// TwinCAT 3 PLC project PLC
// ProgramVersion: 3.1.4023.0
// libraries:
//   Tc2_MC2, * (Beckhoff Automation GmbH)
//   Tc2_Standard, * (Beckhoff Automation GmbH)
//   Tc2_System, * (Beckhoff Automation GmbH)
//   Tc3_Module, * (Beckhoff Automation GmbH)
//   VisuSymbols,3.5.10.0,System
// project tree:
//   DUTs/ E_Axis.TcDUT, E_MachineState.TcDUT, E_Speed.TcDUT, ST_ErrorData.TcDUT
//   / GlobalTextList.TcGTLO, PlcTask.TcTTO, Visualization Manager.TcVMO (not stored), VISU_TASK.TcTTO
//   GVLs/ GVL.TcGVL
//   POUs/ FB_Machine.TcPOU, FB_Tower.TcPOU, F_HeaderErrorMessage.TcPOU, F_NcErrorMessage.TcPOU, MAIN.TcPOU
//   VISUs/ Tower1.TcVIS
// real-time tasks:
//   TASK PlcTask: cycle T#10ms, priority 20, ADS port 350
//   TASK VISU_TASK: cycle T#200000us, priority 30, ADS port 351
// motion (NC):
//   TASK NC-Task 1 SAF: cycle T#2ms, priority 4, ADS port 501
//   TASK NC-Task 1 SVB: cycle T#10ms, priority 8, ADS port 511
//   AXIS Axis 1 (id 1)
//     General: UnitName=m
//     Dynamic: AccelerationMaximum=1.5, DecelerationMaximum=1.5, Acceleration=1.5, Deceleration=1.5, Jerk=2.25
//     Velo: RefSearch=0.03, RefSync=0.03, SlowManual=0.1, FastManual=1, Maximum=0.1
//     OtherSettings: AllowMotionCmdToSlave=true, PulseDistancePos=0.005, PulseDistanceNeg=0.005
//     encoder EncType=1
//       EncPara: ScaleFactorNumerator=4.166666667e-06, ReferenceSystem=1
//         SoftEndMinControl: Enable=true
//         SoftEndMaxControl: Enable=true, Range=1.44
//         TimeComp: TimeCompMode=1, EncDelayCycles=4
//     drive DrvType=5
//       Analog: VeloReferenz=0.416666666666667, TorqueSetpointScale=10, ScaleFactorActTorque=0.1
//       TimeComp: TaskDelayCycles=1
//     controller CtrType=1
//       CtrPara: PriorControlFactor=1
//         Observer: BandWidth=20
// I/O:
//   DEVICE Device 1 (EtherCAT) (disabled), AmsNetId 192.168.100.90.2.1
//     Drive 1 (N5-2-1) [N5 EtherCAT Drive (CoE)]
// variable links:
//   __THIS__ <-> PLC/PLC Instance
//     Inputs/FromPlc <-> PlcTask Outputs/MAIN.Machine.Tower.stAxis.PlcToNc
//     Outputs/ToPlc <-> PlcTask Inputs/MAIN.Machine.Tower.stAxis.NcToPlc
//   __THIS__ <-> Device 1 (EtherCAT)/Drive 1 (N5-2-1)
//     Drive/Inputs/In/nState1 <-> Transmit PDO 1 Mapping Parameter/Statusword
//     Drive/Inputs/In/nState2 <-> Transmit PDO 1 Mapping Parameter/Statusword @bit 8
//     Drive/Inputs/In/nState4 @bit 1 <-> WcState/InputToggle
//     Drive/Inputs/In/nState4 <-> WcState/WcState
//     Drive/Inputs/In/nState5 <-> Transmit PDO 1 Mapping Parameter/Modes of operation display
//     Drive/Outputs/Out/nCtrl1 <-> Receive PDO 1 Mapping Parameter/Controlword
//     Drive/Outputs/Out/nCtrl2 <-> Receive PDO 1 Mapping Parameter/Controlword @bit 8
//     Drive/Outputs/Out/nCtrl5 <-> Receive PDO 1 Mapping Parameter/Modes of operation
//     Drive/Outputs/Out/nDataOut1 <-> Receive PDO 1 Mapping Parameter/Target Position
//     Enc/Inputs/In/nDataIn1 <-> Transmit PDO 1 Mapping Parameter/Position actual value
//     Enc/Inputs/In/nState4 @bit 1 <-> WcState/InputToggle
//     Enc/Inputs/In/nState4 <-> WcState/WcState
//   NC-Task 1 SAF/Axes/Axis 1 <-> PLC/PLC Instance
//     Inputs/FromPlc <-> PlcTask Outputs/MAIN.Machine.Tower.stAxis.PlcToNc
//     Outputs/ToPlc <-> PlcTask Inputs/MAIN.Machine.Tower.stAxis.NcToPlc

CONFIGURATION PLC
    RESOURCE PLC ON TwinCAT3
        TASK PlcTask(INTERVAL := T#10ms, PRIORITY := 20);
        TASK VISU_TASK(INTERVAL := T#200000us, PRIORITY := 30);
        PROGRAM MAIN WITH PlcTask : MAIN;
        PROGRAM VisuElems_Visu_Prg WITH VISU_TASK : VisuElems.Visu_Prg;
    END_RESOURCE
END_CONFIGURATION

// ---- DUTs/E_Axis.TcDUT
{attribute 'qualified_only'}
{attribute 'strict'}
{attribute 'to_string'}
TYPE E_Axis :
(
	Disabled,
	Enabled,
	Idle,
	MoveAbs,
	Stop,
	Error,
	Reset,
	ManualMode
);
END_TYPE

// ---- DUTs/E_MachineState.TcDUT
{attribute 'qualified_only'}
{attribute 'strict'}
{attribute 'to_string'}
TYPE E_MachineState :
(
	Error,
	Ready,
	Running
);
END_TYPE

// ---- DUTs/E_Speed.TcDUT
{attribute 'qualified_only'}
{attribute 'strict'}
{attribute 'to_string'}
TYPE E_Speed :
(
	Low,
	High
);
END_TYPE

// ---- DUTs/ST_ErrorData.TcDUT
TYPE ST_ErrorData :
STRUCT
	nErrorID			: UDINT;
	sTimeStamp			: STRING;
	sErrorMessageBody	: STRING[300];
	sErrorMessageHeader	: STRING[300];	
	eLastState			: E_Axis;
END_STRUCT
END_TYPE

// ---- GVLs/GVL.TcGVL
VAR_GLOBAL

	eMachineState					: E_MachineState;
	UI_EnableHighSpeed				: BOOL;
END_VAR

// ---- POUs/MAIN.TcPOU
PROGRAM MAIN
VAR
	Machine : FB_Machine; 
	
END_VAR

Machine();

END_PROGRAM

// ---- POUs/FB_Machine.TcPOU
FUNCTION_BLOCK FB_Machine
VAR_INPUT
END_VAR
VAR_OUTPUT

END_VAR
VAR
	Tower : FB_Tower;
	//fManualLowSpeed		: LREAL;
	//fManualHighSpeed	: LREAL;	
	
END_VAR

Tower();

(*
MCJog( Axis := 	stAxis, Velocity := fManualVelocity, Mode := MC_JOGMODE_CONTINOUS );				
McPower(Axis := stAxis);
McReset(Axis := stAxis); 
ActUpdateAxisData();
ActUpdateManVelocity();


CASE GVL.eMachineState OF
	

	// The machine starts up in Error state
	E_MachineState.Error:	
	
	// Changes statet to Ready state
	IF startButton THEN
		readyLamp := TRUE;
		SetState( E_MachineState.Ready );
	END_IF
	
	
	
	E_MachineState.Ready:
	McReset.Execute := TRUE;
		IF McReset.Done THEN 
			McReset.Execute := FALSE; 
		END_IF 	
	
		IF (ActualPos < lowerLimit OR ActualPos > upperLimit) AND enableButton THEN
			 
			IF ActualPos > upperLimit AND enableButton THEN
				McPower.Enable 			:= TRUE;
				McPower.Enable_Negative := TRUE;
				SetState( E_MachineState.Running );
			END_IF
			
			IF ActualPos < lowerLimit AND enableButton THEN 
				McPower.Enable 			:= TRUE;
				McPower.Enable_Positive := TRUE;
				SetState( E_MachineState.Running );
			END_IF
		END_IF
		
 		// Enables the axis for movement
		IF enableButton AND ActualPos > lowerLimit AND ActualPos < upperLimit  THEN
			McPower.Enable 			:= TRUE;
			McPower.Enable_Positive := TRUE; 
			McPower.Enable_Negative := TRUE;		
			SetState( E_MachineState.Running );
		END_IF
		
		// Disables the axis for movement
		IF stopButton THEN
			McPower.Enable 			:= FALSE;
			McPower.Enable_Positive := FALSE; 
			McPower.Enable_Negative := FALSE;
			enableButton 			:= FALSE;
			MCJog.JogForward 		:= FALSE; 
			MCJog.JogBackwards 		:= FALSE;
		END_IF
			
			
	E_MachineState.Running: 	
		
		// forward and backward movement logic
		IF forwardButton OR backwardButton THEN
			IF (ActualPos > lowerLimit AND ActualPos < upperLimit) THEN 
				McPower.Enable_Positive := TRUE; 
				McPower.Enable_Negative := TRUE;
			END_IF 
			IF forwardButton THEN 
				MCJog.JogForward 	:= TRUE;
				MCJog.JogBackwards 	:= FALSE;
			END_IF 
			
			IF backwardButton THEN
				MCJog.JogBackwards 	:= TRUE; 
				MCJog.JogForward 	:= FALSE;
			END_IF 
		ELSE 
			MCJog.JogBackwards 	:= FALSE;
			MCJog.JogForward 	:= FALSE;
		END_IF
		
		// Disables the axis for movement
		IF stopButton THEN
			McPower.Enable 			:= FALSE;
			McPower.Enable_Positive := FALSE; 
			McPower.Enable_Negative := FALSE;
			enableButton 			:= FALSE;
			MCJog.JogForward 		:= FALSE; 
			MCJog.JogBackwards 		:= FALSE;
	
			SetState( E_MachineState.Ready );
		END_IF  
		
		IF (ActualPos < lowerLimit OR ActualPos > upperLimit) AND McPower.Enable_Positive AND McPower.Enable_Negative THEN 
			McPower.Enable 			:= FALSE;
			McPower.Enable_Positive := FALSE; 
			McPower.Enable_Negative := FALSE;
			enableButton 			:= FALSE;
			MCJog.JogForward 		:= FALSE; 
			MCJog.JogBackwards 		:= FALSE;
	
			SetState( E_MachineState.Error );
		END_IF
		

END_CASE

*)

END_FUNCTION_BLOCK

// ---- POUs/FB_Tower.TcPOU

FUNCTION_BLOCK FB_Tower
VAR_INPUT
	resetButton			: BOOL;
	startButton			: BOOL;
	stopButton 			: BOOL;
	forwardButton 		: BOOL; 
	backwardButton 		: BOOL;
	fManualVelocity		: LREAL;
	
	// velocity constant for HIGH and LOW value. 
	fManualLowSpeed		: LREAL := 0.05;
	fManualHighSpeed	: LREAL := 0.1;	
END_VAR
VAR_OUTPUT
END_VAR
VAR
	// Libraries used
	stAxis 				: AXIS_REF;
	MCJog 				: MC_Jog;
	McPower 			: MC_Power;
	McReset				: MC_Reset;
	stErrorData			: ST_ErrorData; 
	
	// Real axis data feedback
	Enabled     		: BOOL;
	ActualVel   		: LREAL;
	ActualPos  			: LREAL;
	
	//ActualTorque		: LREAL; 
	bPositiveDirection	: BOOL; 
	bNegativeDirection	: BOOL;
	AxisMovement		: BOOL; 
	bMinSoftLimit		: BOOL;
	bMaxSoftLimit		: BOOL; 
	
	// Error id 
	mc_errorID 			: UDINT := 1; 
	mc_error_string 	: STRING; 
	error_header_string	: STRING;
	
	// For blinking lamp
	light_pulse 		: BOOL; 
	light_constant 		: BOOL; 
	tBlink 				: TON; 
	blink1000 			: BOOL;
	
	//Adjusting speed on axis
	SpeedSetting		: E_Speed; 
	
	// TO_STRING for velocity 

	ESpeed         		: E_Speed;
    nCurrentValue   	: INT;
    sCurrentValue   	: STRING;
    wsCurrentValue  	: WSTRING;
    sComponent      	: STRING;
    wsComponent     	: WSTRING;
	
	// TO_STRING for states
	EMachineState 		: E_MachineState;
	nCurrentState   	: INT;
	sCurrentState		: STRING;
	wsCurrentState		: WSTRING;
	sComponentState		: STRING;
	wsComponentState	: WSTRING;
	
	{IF defined (Emulation)}
	StateTower1					AT %I* : UINT := 8;
	{ELSE}
	StateTower1					AT %I* : UINT;
	{END_IF}
END_VAR

MCJog( Axis := 	stAxis, Velocity := fManualVelocity, Mode := MC_JOGMODE_CONTINOUS );				
McPower(Axis := stAxis);
McReset(Axis := stAxis); 
ActUpdateAxisData();
ActUpdateManVelocity();
ActBlinkingTimer(); 
ActToStringSpeedAndState();
CASE GVL.eMachineState OF
	
	// The machine starts up in Error state
	E_MachineState.Error:	
	
	light_constant := FALSE;
	EnableAxis(FALSE);
	mc_error_string := F_NcErrorMessage(mc_errorID);
	error_header_string := F_HeaderErrorMessage(mc_errorID);

	IF resetButton THEN
		SetState( E_MachineState.Ready );
	END_IF
	
	// Ready state is for enabling the axis
	E_MachineState.Ready:
	light_constant := FALSE;
	McResetAxis();
	
	IF startButton THEN 
		light_constant := TRUE; 
		EnableAxis(TRUE);
		SetState( E_MachineState.Running );
	END_IF
	
	// Running state is for driving the axis in both postive and negative Y direction. 
	E_MachineState.Running:
	
	MCJog.JogForward 	:= forwardButton; 
	MCJog.JogBackwards 	:= backwardButton;
	
	IF stopButton THEN 
		EnableAxis(FALSE);
		SetState( E_MachineState.Ready );
	END_IF
END_CASE

ACTION ActBlinkingTimer:
tBlink(IN := NOT tblink.Q, PT := T#1S);
blink1000 := tBlink.ET > T#0.5S;

light_pulse := light_constant OR blink1000;
END_ACTION

ACTION ActToStringSpeedAndState:
nCurrentValue := ESpeed; 

sCurrentValue  := TO_STRING(ESpeed); 
wsCurrentValue := TO_WSTRING(ESpeed); 

sComponent     := TO_STRING(E_Speed.High); 
wsComponent    := TO_WSTRING(E_Speed.Low);

nCurrentState := EMachineState;

sCurrentState  := TO_STRING(EMachineState); 
wsCurrentState  := TO_WSTRING(EMachineState); 

sComponentState      := TO_STRING(E_MachineState.Ready); 
wsComponentState     := TO_WSTRING(E_MachineState.Running);
END_ACTION

ACTION ActUpdateAxisData:
// Data from NC interface
stAxis.ReadStatus();
Enabled      		:= McPower.Status;
ActualPos 			:= stAxis.NcToPlc.ActPos;
ActualVel			:= stAxis.NcToPlc.ActVelo;

//ActualTorque		:= ActualTorqueNm;
bPositiveDirection	:= stAxis.Status.PositiveDirection;
bNegativeDirection	:= stAxis.Status.NegativeDirection;
AxisMovement		:= stAxis.Status.Moving;
bMinSoftLimit		:= stAxis.Status.SoftLimitMinExceeded;
bMaxSoftLimit		:= stAxis.Status.SoftLimitMaxExceeded;
END_ACTION

ACTION ActUpdateManVelocity:
CASE SpeedSetting OF 

	E_Speed.Low:
	
		IF GVL.UI_EnableHighSpeed THEN
			fManualVelocity			:= fManualHighSpeed;
			SpeedSetting			:= E_Speed.High;
			
		ELSE
			fManualVelocity			:= fManualLowSpeed;
		END_IF
	
	E_Speed.High:
	
		IF NOT GVL.UI_EnableHighSpeed THEN
			fManualVelocity			:= fManualLowSpeed;
			SpeedSetting			:= E_Speed.Low;
		ELSE
			fManualVelocity			:= fManualHighSpeed;
		END_IF

END_CASE
END_ACTION

METHOD EnableAxis : BOOL
VAR_INPUT
	axisBoolStatus : BOOL; 
END_VAR
McPower.Enable 			:= axisBoolStatus;
McPower.Enable_Positive := axisBoolStatus;
McPower.Enable_Negative := axisBoolStatus;
END_METHOD

METHOD ErrorUpdate
VAR_INPUT
	eState				: E_Axis;
	nErrorId			: UDINT;
	sErrorMessageBody	: STRING[300];
END_VAR
VAR
	sErrorMessageHeader	: STRING[300];
END_VAR

stErrorData.eLastState			:= eState;
stErrorData.nErrorID			:= nErrorId;
stErrorData.sErrorMessageBody	:= sErrorMessageBody;
stErrorData.sErrorMessageHeader	:= F_HeaderErrorMessage(nErrorId);
END_METHOD

METHOD McResetAxis : BOOL
VAR_INPUT
END_VAR
McReset.Execute := TRUE;

IF McReset.Done THEN 
	McReset.Execute := FALSE; 
END_IF
END_METHOD

METHOD SetState
VAR_INPUT
	eState	: E_MachineState;
END_VAR
GVL.eMachineState	:= eState;
END_METHOD

END_FUNCTION_BLOCK

// ---- POUs/F_NcErrorMessage.TcPOU
FUNCTION F_NcErrorMessage : STRING[2048]
VAR_INPUT
	Error		: UDINT;
END_VAR

CASE Error OF
		0		: 		F_NcErrorMessage	:= 'None';

(* --> User defined errors for entire machine <--*)
		1		:		F_NcErrorMessage	:= 'The machine is in error at startup - please reset. ';		

		ELSE
			IF 36844 < Error AND Error < 36857 THEN
				F_NcErrorMessage:='NC3_Internal_Unexpected INTERNAL Error';
			ELSE		
				F_NcErrorMessage:='Msg Unknown';
			END_IF	

END_CASE

END_FUNCTION

// ---- POUs/F_HeaderErrorMessage.TcPOU
FUNCTION F_HeaderErrorMessage : STRING
VAR_INPUT
	ErrorID		: UDINT;
END_VAR

IF ErrorID = 0 THEN
	F_HeaderErrorMessage := 'None';
ELSIF ErrorID = 1 THEN
	F_HeaderErrorMessage := 'Startup safety';
END_IF

END_FUNCTION

// ---- GlobalTextList.TcGTLO
TEXTLIST GlobalTextList
  242 = ''
  377 = '%1.2f m'
  210 = '%s'
  857 = '------>'
  1232 = '1'
  1699 = '10'
  1682 = '2'
  1336 = '3'
  2102 = '4'
  319 = '5'
  1432 = '6'
  830 = '7'
  1654 = '8'
  887 = '9'
  426 = '<-----'
  989 = 'Axis 1'
  132 = 'Axis 2'
  347 = 'Axis 3'
  348 = 'Axis 4'
  701 = 'Axis 5'
  1208 = 'Back'
  1592 = 'Buffer status'
  1486 = 'Cancel'
  487 = 'Down'
  2786 = 'Empty'
  624 = 'Enable'
  186 = 'ENABLED'
  2871 = 'End Manual Control'
  43 = 'Error'
  723 = 'ERROR'
  1933 = 'Feed out'
  117 = 'Feeding out'
  3026 = 'Full'
  599 = 'Has pallet'
  2256 = 'High'
  2883 = 'Id: %d'
  2487 = 'Last pallet id'
  755 = 'Low'
  265 = 'MACHINE READY'
  345 = 'Main'
  107 = 'MAIN.Machine.Tower.ActualPos'
  679 = 'Manual Control'
  115 = 'Manual Operation Deactivated'
  872 = 'Move left'
  175 = 'MOVE LEFT'
  587 = 'Move right'
  850 = 'MOVE RIGHT'
  2947 = 'Mute'
  3046 = 'No'
  1515 = 'Platform status'
  746 = 'Position'
  201 = 'Ready'
  715 = 'READY'
  91 = 'Reset'
  714 = 'Robot'
  119 = 'RUNNING'
  1248 = 'Show more (%d)'
  937 = 'Speed'
  111 = 'Speed:'
  943 = 'Start'
  135 = 'START'
  589 = 'Start '
  2600 = 'Starting in: %d s'
  463 = 'Status'
  346 = 'Stop'
  805 = 'STOP'
  2202 = 'Testing Disabled'
  938 = 'Testing Enabled'
  1915 = 'Toggle the options to enable/disable axis errors. Once disabled, the axis will ignore all errors, and the machine cannot run autonomously.'
  416 = 'Tower 1'
  461 = 'Tower 10'
  206 = 'Tower 2'
  567 = 'Tower 3'
  419 = 'Tower 4'
  65 = 'Tower 5'
  153 = 'Tower 6'
  774 = 'Tower 7'
  133 = 'Tower 8'
  940 = 'Tower 9'
  350 = 'Towers'
  86 = 'TURN ON MACHINE'
  134 = 'Unmute'
  705 = 'Up'
  2770 = 'Yes'
  1960 = '‹'
  1985 = '›'
END_TEXTLIST

// ---- VISUs/Tower1.TcVIS
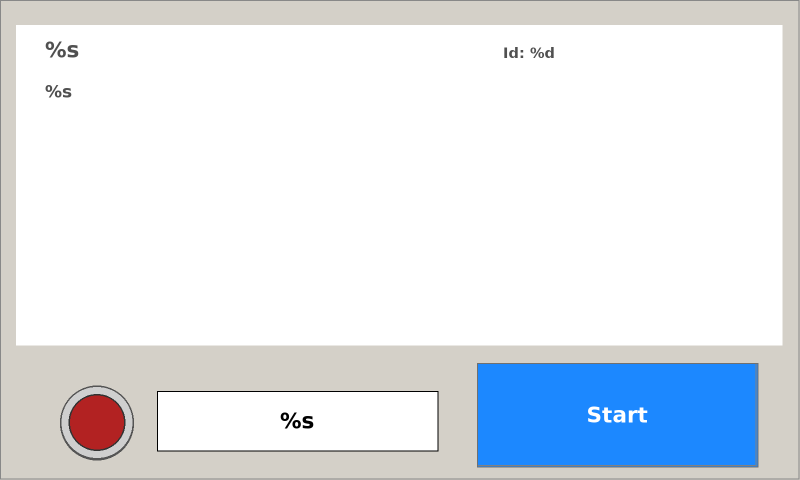
VISUALIZATION Tower1  // 800x480
    Button (110,230 150x110), "Down"
    Button (110,90 150x110), "Up"
    Button (110,90 150x110), "Up", invisible if: NOT(MAIN.Machine.Tower.Enabled)
        tap MAIN.Machine.Tower.backwardButton
    Button (110,230 150x110), "Down", invisible if: GVL.eMachineState = E_MachineState.Error OR NOT(MAIN.Machine.Tower.Enabled)
        tap MAIN.Machine.Tower.forwardButton
    Rectangle (608,99 110x50), "Low", invisible if: GVL.UI_EnableHighSpeed = False
        toggle GVL.UI_EnableHighSpeed
    Rectangle (608,99 110x50), "High", invisible if: GVL.eMachineState = E_MachineState.Error or GVL.UI_EnableHighSpeed = True
        toggle GVL.UI_EnableHighSpeed
    Label (2039,520 94x27), "Position", invisible if: GVL.eMachineState = E_MachineState.Error
    RoundedRectangle (2039,555 137x23), "%1.2f m", text variable: MAIN.Machine.Tower.ActualPos, invisible if: GVL.eMachineState = E_MachineState.Error
    Label (459,79 139x27), "Speed:"
    RoundedRectangle (460,109 96x36), "%s", text variable: TO_STRING(MAIN.Machine.Tower.SpeedSetting)
    Lamp1 (45,381 104x85), variable: MAIN.Machine.Tower.light_pulse, invisible if: GVL.eMachineState = E_MachineState.Error, style: Lamp-Lamp1-Green
    RoundedRectangle (157,391 281x60), "%s", text variable: TO_STRING(GVL.eMachineState)
    Button (477,363 281x104), "Stop", invisible if: GVL.eMachineState = E_MachineState.Error OR GVL.eMachineState = E_MachineState.Ready
        tap MAIN.Machine.Tower.stopButton
    Lamp1 (45,380 104x85), variable: MAIN.Machine.Tower.light_pulse, invisible if: NOT(GVL.eMachineState = E_MachineState.Error), style: Lamp-Lamp1-Red
    Button (477,363 281x104), "Reset", invisible if: NOT(GVL.eMachineState = E_MachineState.Error)
        tap MAIN.Machine.Tower.resetButton
    Button (477,363 281x104), "Start", invisible if: GVL.eMachineState = E_MachineState.Error OR MAIN.Machine.Tower.Enabled OR MAIN.Machine.Tower.Enabled
        tap MAIN.Machine.Tower.startButton
    Rectangle (16,25 766x320), invisible if: NOT(GVL.eMachineState = E_MachineState.Error)
    Rectangle (42,80 600x105), "%s", text variable: MAIN.Machine.Tower.mc_error_string, invisible if: NOT(GVL.eMachineState = E_MachineState.Error)
    Rectangle (42,27 452x46), "%s", text variable: MAIN.Machine.Tower.error_header_string, invisible if: NOT(GVL.eMachineState = E_MachineState.Error)
    Rectangle (500,30 136x46), "Id: %d", text variable: MAIN.Machine.Tower.mc_errorID, invisible if: NOT(GVL.eMachineState = E_MachineState.Error)
END_VISUALIZATION
